INTERFACE I_XTS_Mover EXTENDS __SYSTEM.IQueryInterface

{attribute 'OPC.UA.DA.Property' := '1'}
{attribute 'monitoring':='call'}
PROPERTY Coupled : BOOL
GET
END_GET
END_PROPERTY

METHOD Disable : HRESULT
VAR_INPUT
END_VAR
END_METHOD

{attribute 'monitoring':='call'}
PROPERTY DrivenDistance : LREAL
GET
END_GET
END_PROPERTY

METHOD Enable : HRESULT
VAR_INPUT
END_VAR
END_METHOD

{attribute 'OPC.UA.DA.Property' := '1'}
{attribute 'monitoring':='call'}
PROPERTY Feedback : I_CH_Feedback
GET
END_GET
END_PROPERTY

PROPERTY getAxisRef : REFERENCE TO Tc2_MC2.AXIS_REF
GET
END_GET
END_PROPERTY

METHOD HaltCA : HRESULT
VAR_INPUT
END_VAR
END_METHOD

{attribute 'monitoring':='call'}
PROPERTY IdentInGroup : IDENT_IN_GROUP_REF
GET
END_GET
END_PROPERTY

{attribute 'monitoring':='call'}
PROPERTY LagDistance : LREAL
GET
END_GET
END_PROPERTY

{attribute 'monitoring':='call'}
PROPERTY LastCmdTargedGap : LREAL
GET
END_GET
END_PROPERTY

{attribute 'monitoring':='call'}
PROPERTY LastCmdTargedPosition : LREAL
GET
END_GET
END_PROPERTY

{attribute 'monitoring':='call'}
PROPERTY LastCmdTargedVelocity : LREAL
GET
END_GET
END_PROPERTY

METHOD MoveAbsCA : HRESULT
VAR_INPUT
    fPosition              : LREAL;
    fVelocity              : LREAL;
    fGap                   : LREAL;
    eDirection             : Tc3_Mc3Definitions.MC_DIRECTION;
END_VAR
END_METHOD

{attribute 'monitoring':='call'}
PROPERTY MoverInGroup : BOOL
GET
END_GET
SET
END_SET
END_PROPERTY

{attribute 'OPC.UA.DA.Property' := '1'}
{attribute 'monitoring':='call'}
PROPERTY Moving : BOOL
GET
END_GET
END_PROPERTY

{attribute 'monitoring':='call'}
PROPERTY NextMover : I_XTS_Mover
GET
END_GET
END_PROPERTY

{attribute 'monitoring':='call'}
PROPERTY OID : OTCID
GET
END_GET
END_PROPERTY

{attribute 'monitoring':='call'}
PROPERTY ParentStation : I_XTS_Station
GET
END_GET
SET
END_SET
END_PROPERTY

{attribute 'monitoring':='call'}
PROPERTY PositionOnTrack : LREAL
GET
END_GET
END_PROPERTY

METHOD Reset : HRESULT
VAR_INPUT
END_VAR
END_METHOD

{attribute 'monitoring':='call'}
PROPERTY SetAcceleration : LREAL
GET
END_GET
END_PROPERTY

{attribute 'monitoring':='call'}
PROPERTY SetVelocity : LREAL
GET
END_GET
END_PROPERTY

{attribute 'monitoring':='call'}
PROPERTY TargedStation : STRING
GET
END_GET
SET
END_SET
END_PROPERTY

{attribute 'monitoring':='call'}
PROPERTY UtilityMover : I_TcIoXtsXpuMover
GET
END_GET
END_PROPERTY

END_INTERFACE

(* stored: Version 1.1.0.1, ProductVersion 3.1.4024.12
   Itf I_XTS_Mover: Id {5e8caa86-9ac3-4695-8c34-e1bf5bc823f4}
   Property Coupled: Id {f139e77a-7c2a-489e-91ef-49f7b2e94bba}
   Get Get: Id {faae7b28-3b09-4cf5-ab4e-56e7824857e7}
   Method Disable: Id {b6456993-11bc-494c-812d-d6ee15dd15d3}
   Property DrivenDistance: Id {bb4a8d98-2f04-4ac5-8f87-fb9810e9f0a0}
   Get Get: Id {b214eab2-7548-4cd2-8e4a-70d4c034ee1b}
   Method Enable: Id {1299f19e-8449-4a27-8d5f-f0a4ec5ea67d}
   Property Feedback: Id {092eee79-82dc-442c-affb-0dda1f3ce08e}
   Get Get: Id {4b630cec-61a7-45de-b605-2fcfc3fc8ed0}
   Property getAxisRef: Id {7d704c79-9177-4837-abc3-f85effa85ad8}
   Get Get: Id {bab85460-ac62-4e5a-9c6c-e4dfec154c6e}
   Method HaltCA: Id {a6ecf43b-3167-42c5-81bc-d764b9843f91}
   Property IdentInGroup: Id {41501d47-ce1d-4dee-bad9-a6c403b1fb91}
   Get Get: Id {b9838914-b19f-441b-ad0f-3c63f1055bc7}
   Property LagDistance: Id {9a2c68cf-4180-4c4b-9d8e-db768a5fdfc9}
   Get Get: Id {0f1c7692-616b-42d5-a98a-0594c911dcd9}
   Property LastCmdTargedGap: Id {67b3f9aa-9989-47de-ade8-aec428c65ae0}
   Get Get: Id {9d0b0751-4159-40a8-a6dd-8a9fc36ca3ea}
   Property LastCmdTargedPosition: Id {acd15eb0-4349-4e9e-846c-32369b16a3c2}
   Get Get: Id {0e298aa1-f441-47b4-9dfa-510d2add6c83}
   Property LastCmdTargedVelocity: Id {4811ac25-c82a-4a7a-aa8e-b7de97e686c0}
   Get Get: Id {a4f40d54-e4e1-4d35-943e-ed0f94de41d0}
   Method MoveAbsCA: Id {b04f4e40-9816-4b26-bc86-b6d5bb1e599c}
   Property MoverInGroup: Id {fe32ef80-0d8e-45c4-9bd0-c5f7c8e7c4aa}
   Get Get: Id {31c8cdcb-d465-45bf-abe6-f78ba346a881}
   Set Set: Id {9bab0b75-4ef9-4b96-9c54-1519bf62a981}
   Property Moving: Id {ae4a6134-73ca-4cf9-837a-70d7fa340c28}
   Get Get: Id {63ee907c-8cb1-4861-a6e6-cec4bf3019b5}
   Property NextMover: Id {decab6a5-ffa7-4e0a-b90d-4597d5401c33}
   Get Get: Id {d0b0fc82-1e96-41f3-94ef-e9497b2c44e9}
   Property OID: Id {ba060d70-1ddd-4572-b02f-fa56abbd4565}
   Get Get: Id {40b2a673-3213-4794-8446-65dfcdaff142}
   Property ParentStation: Id {e9ff5c0c-0ed5-4fed-b169-133939b76103}
   Get Get: Id {b4cfe583-61a8-4b9e-8938-43b6ad0bbf8b}
   Set Set: Id {ab4415ee-b659-4dd7-8fae-c92384b39427}
   Property PositionOnTrack: Id {9e9eca9f-dcb1-4b0f-9cfd-58ac01185b57}
   Get Get: Id {0d4004f2-f5ee-44b1-b172-96d1b9fb4bc3}
   Method Reset: Id {3072dcd8-03bd-4211-a2f3-28efc2657689}
   Property SetAcceleration: Id {0aa41afe-225c-4fc1-9438-f89f5c85e45b}
   Get Get: Id {0d57e38c-f19b-4df3-9348-5d9762a1a333}
   Property SetVelocity: Id {eca871ef-3259-414d-9ab1-8eda8911327b}
   Get Get: Id {8a016fe7-9be9-493b-823c-bc13acf41b15}
   Property TargedStation: Id {aeef0653-da7a-4e18-bc90-04feb4afd3d6}
   Get Get: Id {4cb8dd61-c282-4bdd-965f-750f10d5d022}
   Set Set: Id {c3126502-78ae-4e98-beb4-8531e11c8d9e}
   Property UtilityMover: Id {699d7538-c532-42d1-9a3b-a8ada9f2a844}
   Get Get: Id {8a4555b4-c54b-44e8-b201-9974e9eacb64} *)
